Yaskawa INFORM job: SPINDE_AIR_OFF.JBI

/JOB
//NAME SPINDE_AIR_OFF
//POS
///NPOS 0,0,0,0,0,0
//INST
///DATE 2022/03/01 16:25
///ATTR SC,RW
///GROUP1 RB1
NOP
DOUT OT#(17) OFF
END
